Staubli VAL3: Day1.pjx

--- Day1.pjx ---
Parameters version=s8.13.1Cs9_BS2800 stackSize=5000 millimeterUnit=true
Program file=start.pgx
Program file=stop.pgx
Data file=Day1.dtx
Library alias=math path=Disk://math/math.pjx
Library alias=util path=Disk://helpers/helpers.pjx

--- Day1.dtx ---
num nVector[10]
num nResult
string sInput
num nResult2
bool bResult
num nInput

--- start.pgx ---
program start()
begin

  // read file
  call util:readFile("Disk://input_day1.txt", sInput)

  // PUZZLE 1
  // vec2num
  call util:vec2num(sInput, nInput)

  // calc diff between elements
  call math:diff(nInput, nResult2)

  // compare elements if step is >0
  call util:compare(nResult2, ">", 0, bResult)

  // count steps > 0
  call util:countBool(bResult, nResult)
  ? nResult

  // PUZZLE 2
  call math:rollsum(nInput, 3, nResult)

  // calc diff between elements
  call math:diff(nResult, nResult2)

  // compare elements if step is >0
  call util:compare(nResult2, ">", 0, bResult)

  // count steps > 0
  call util:countBool(bResult, nResult)
  ? nResult

end

--- stop.pgx ---
program stop()
begin

end
